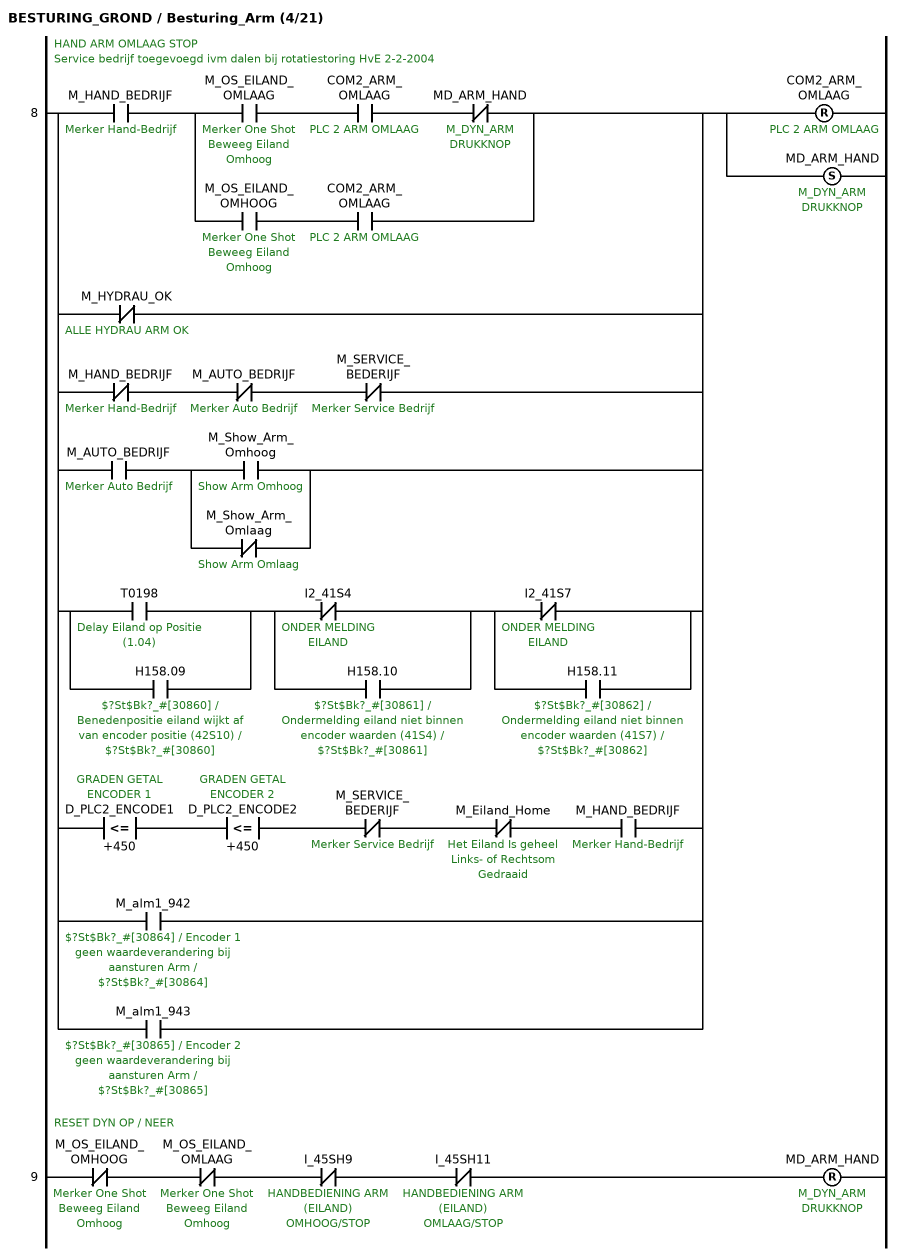
; [picture p373: BESTURING_GROND / Besturing_Arm, rungs 8-9]
; rung 8: HAND ARM OMLAAG STOP / Service bedrijf toegevoegd ivm dalen bij rotatiestoring HvE 2-2-2004
LD M_HAND_BEDRIJF  ; Merker Hand-Bedrijf
LD M_OS_EILAND_OMLAAG  ; Merker One Shot Beweeg Eiland Omhoog
AND COM2_ARM_OMLAAG  ; PLC 2 ARM OMLAAG
ANDNOT MD_ARM_HAND  ; M_DYN_ARM DRUKKNOP
LD M_OS_EILAND_OMHOOG  ; Merker One Shot Beweeg Eiland Omhoog
AND COM2_ARM_OMLAAG  ; PLC 2 ARM OMLAAG
ORLD
ANDLD
ORNOT M_HYDRAU_OK  ; ALLE HYDRAU ARM OK
LDNOT M_HAND_BEDRIJF  ; Merker Hand-Bedrijf
ANDNOT M_AUTO_BEDRIJF  ; Merker Auto Bedrijf
ANDNOT M_SERVICE_BEDERIJF  ; Merker Service Bedrijf
ORLD
LD M_AUTO_BEDRIJF  ; Merker Auto Bedrijf
LD M_Show_Arm_Omhoog  ; Show Arm Omhoog
ORNOT M_Show_Arm_Omlaag  ; Show Arm Omlaag
ANDLD
ORLD
LD T0198  ; Delay Eiland op Positie (1.04)
OR H158.09  ; $?St$Bk?_#[30860] / Benedenpositie eiland wijkt af van encoder positie (42S10) / $?St$Bk?_#[30860]
LDNOT I2_41S4  ; ONDER MELDING EILAND
OR H158.10  ; $?St$Bk?_#[30861] / Ondermelding eiland niet binnen encoder waarden (41S4) / $?St$Bk?_#[30861]
ANDLD
LDNOT I2_41S7  ; ONDER MELDING EILAND
OR H158.11  ; $?St$Bk?_#[30862] / Ondermelding eiland niet binnen encoder waarden (41S7) / $?St$Bk?_#[30862]
ANDLD
ORLD
LD<=S(317) D_PLC2_ENCODE1 +450  ; GRADEN GETAL ENCODER 1
AND<=S(317) D_PLC2_ENCODE2 +450  ; GRADEN GETAL ENCODER 2
ANDNOT M_SERVICE_BEDERIJF  ; Merker Service Bedrijf
ANDNOT M_Eiland_Home  ; Het Eiland Is geheel Links- of Rechtsom Gedraaid
AND M_HAND_BEDRIJF  ; Merker Hand-Bedrijf
ORLD
OR M_alm1_942  ; $?St$Bk?_#[30864] / Encoder 1 geen waardeverandering bij aansturen Arm / $?St$Bk?_#[30864]
OR M_alm1_943  ; $?St$Bk?_#[30865] / Encoder 2 geen waardeverandering bij aansturen Arm / $?St$Bk?_#[30865]
RSET COM2_ARM_OMLAAG  ; PLC 2 ARM OMLAAG
SET MD_ARM_HAND  ; M_DYN_ARM DRUKKNOP
; rung 9: RESET DYN OP / NEER
LDNOT M_OS_EILAND_OMHOOG  ; Merker One Shot Beweeg Eiland Omhoog
ANDNOT M_OS_EILAND_OMLAAG  ; Merker One Shot Beweeg Eiland Omhoog
ANDNOT I_45SH9  ; HANDBEDIENING ARM (EILAND) OMHOOG/STOP
ANDNOT I_45SH11  ; HANDBEDIENING ARM (EILAND) OMLAAG/STOP
RSET MD_ARM_HAND  ; M_DYN_ARM DRUKKNOP

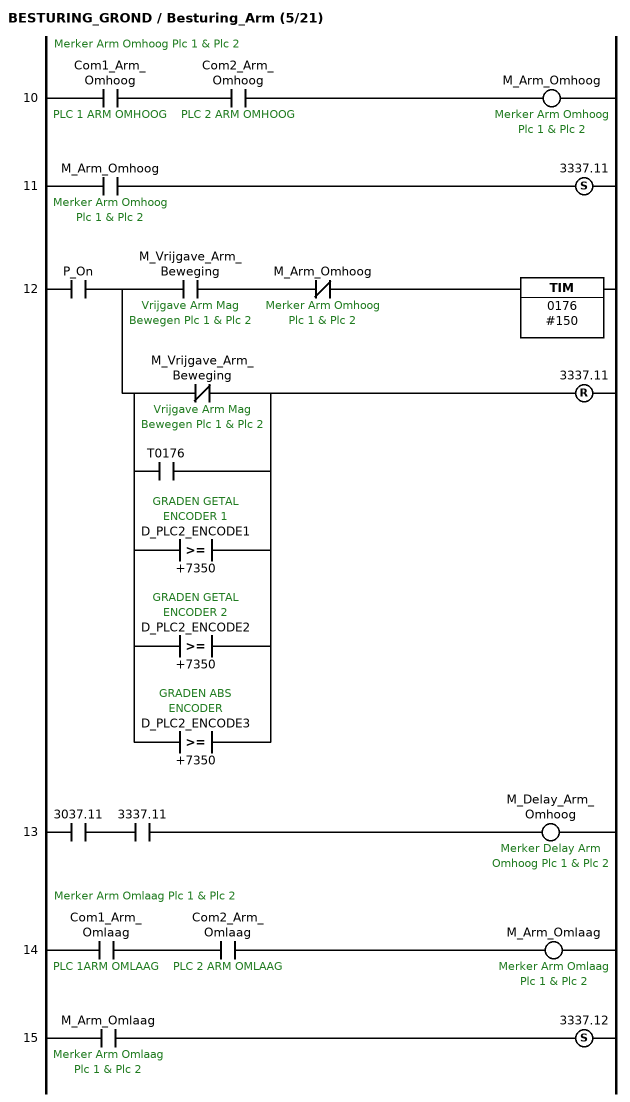
; rung 10: Merker Arm Omhoog Plc 1 & Plc 2
LD Com1_Arm_Omhoog  ; PLC 1 ARM OMHOOG
AND Com2_Arm_Omhoog  ; PLC 2 ARM OMHOOG
OUT M_Arm_Omhoog  ; Merker Arm Omhoog Plc 1 & Plc 2
; rung 11
LD M_Arm_Omhoog  ; Merker Arm Omhoog Plc 1 & Plc 2
SET 3337.11
; rung 12
LD P_On
OUT TR0
AND M_Vrijgave_Arm_Beweging  ; Vrijgave Arm Mag Bewegen Plc 1 & Plc 2
ANDNOT M_Arm_Omhoog  ; Merker Arm Omhoog Plc 1 & Plc 2
TIM 0176 #150
LD TR0
LDNOT M_Vrijgave_Arm_Beweging  ; Vrijgave Arm Mag Bewegen Plc 1 & Plc 2
OR T0176
OR>=S(327) D_PLC2_ENCODE1 +7350  ; GRADEN GETAL ENCODER 1
OR>=S(327) D_PLC2_ENCODE2 +7350  ; GRADEN GETAL ENCODER 2
OR>=S(327) D_PLC2_ENCODE3 +7350  ; GRADEN ABS ENCODER
ANDLD
RSET 3337.11
; rung 13
LD 3037.11
AND 3337.11
OUT M_Delay_Arm_Omhoog  ; Merker Delay Arm Omhoog Plc 1 & Plc 2
; rung 14: Merker Arm Omlaag Plc 1 & Plc 2
LD Com1_Arm_Omlaag  ; PLC 1ARM OMLAAG
AND Com2_Arm_Omlaag  ; PLC 2 ARM OMLAAG
OUT M_Arm_Omlaag  ; Merker Arm Omlaag Plc 1 & Plc 2
; rung 15
LD M_Arm_Omlaag  ; Merker Arm Omlaag Plc 1 & Plc 2
SET 3337.12

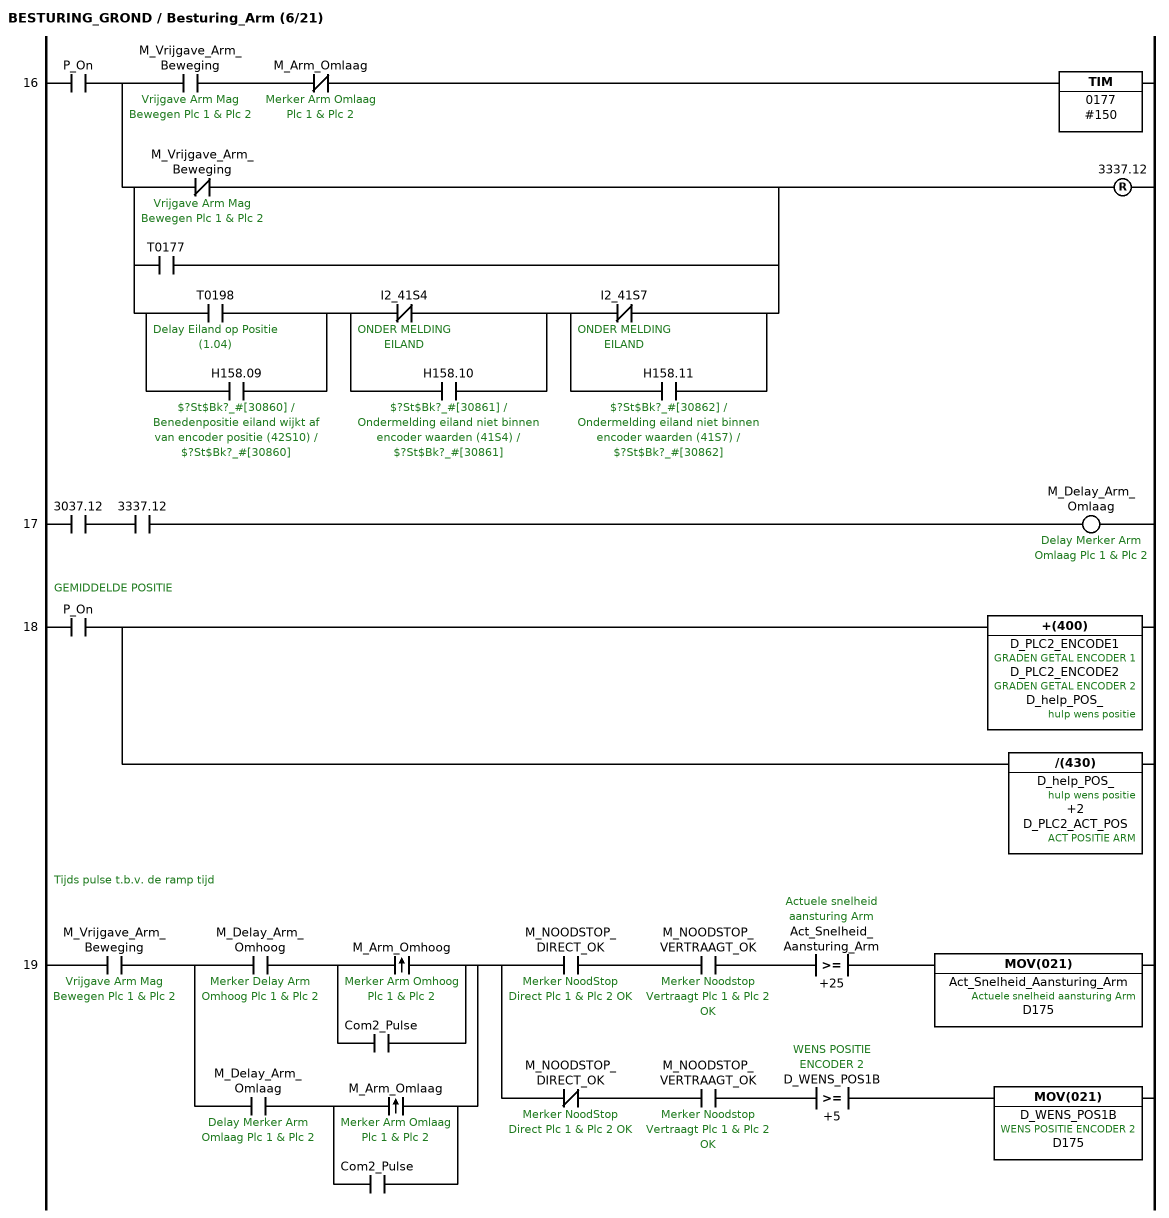
; rung 16
LD P_On
OUT TR0
AND M_Vrijgave_Arm_Beweging  ; Vrijgave Arm Mag Bewegen Plc 1 & Plc 2
ANDNOT M_Arm_Omlaag  ; Merker Arm Omlaag Plc 1 & Plc 2
TIM 0177 #150
LD TR0
LDNOT M_Vrijgave_Arm_Beweging  ; Vrijgave Arm Mag Bewegen Plc 1 & Plc 2
OR T0177
LD T0198  ; Delay Eiland op Positie (1.04)
OR H158.09  ; $?St$Bk?_#[30860] / Benedenpositie eiland wijkt af van encoder positie (42S10) / $?St$Bk?_#[30860]
LDNOT I2_41S4  ; ONDER MELDING EILAND
OR H158.10  ; $?St$Bk?_#[30861] / Ondermelding eiland niet binnen encoder waarden (41S4) / $?St$Bk?_#[30861]
ANDLD
LDNOT I2_41S7  ; ONDER MELDING EILAND
OR H158.11  ; $?St$Bk?_#[30862] / Ondermelding eiland niet binnen encoder waarden (41S7) / $?St$Bk?_#[30862]
ANDLD
ORLD
ANDLD
RSET 3337.12
; rung 17
LD 3037.12
AND 3337.12
OUT M_Delay_Arm_Omlaag  ; Delay Merker Arm Omlaag Plc 1 & Plc 2
; rung 18: GEMIDDELDE POSITIE
LD P_On
+(400) D_PLC2_ENCODE1 D_PLC2_ENCODE2 D_help_POS_  ; GRADEN GETAL ENCODER 1, GRADEN GETAL ENCODER 2, hulp wens positie
/(430) D_help_POS_ +2 D_PLC2_ACT_POS  ; hulp wens positie, ACT POSITIE ARM
; rung 19: Tijds pulse t.b.v. de ramp tijd
LD M_Vrijgave_Arm_Beweging  ; Vrijgave Arm Mag Bewegen Plc 1 & Plc 2
LD M_Delay_Arm_Omhoog  ; Merker Delay Arm Omhoog Plc 1 & Plc 2
@LD M_Arm_Omhoog  ; Merker Arm Omhoog Plc 1 & Plc 2
OR Com2_Pulse
ANDLD
LD M_Delay_Arm_Omlaag  ; Delay Merker Arm Omlaag Plc 1 & Plc 2
@LD M_Arm_Omlaag  ; Merker Arm Omlaag Plc 1 & Plc 2
OR Com2_Pulse
ANDLD
ORLD
ANDLD
OUT TR0
AND M_NOODSTOP_DIRECT_OK  ; Merker NoodStop Direct Plc 1 & Plc 2 OK
AND M_NOODSTOP_VERTRAAGT_OK  ; Merker Noodstop Vertraagt Plc 1 & Plc 2 OK
AND>=S(327) Act_Snelheid_Aansturing_Arm +25  ; Actuele snelheid aansturing Arm
MOV(021) Act_Snelheid_Aansturing_Arm D175  ; Actuele snelheid aansturing Arm
LD TR0
ANDNOT M_NOODSTOP_DIRECT_OK  ; Merker NoodStop Direct Plc 1 & Plc 2 OK
AND M_NOODSTOP_VERTRAAGT_OK  ; Merker Noodstop Vertraagt Plc 1 & Plc 2 OK
AND>=S(327) D_WENS_POS1B +5  ; WENS POSITIE ENCODER 2
MOV(021) D_WENS_POS1B D175  ; WENS POSITIE ENCODER 2

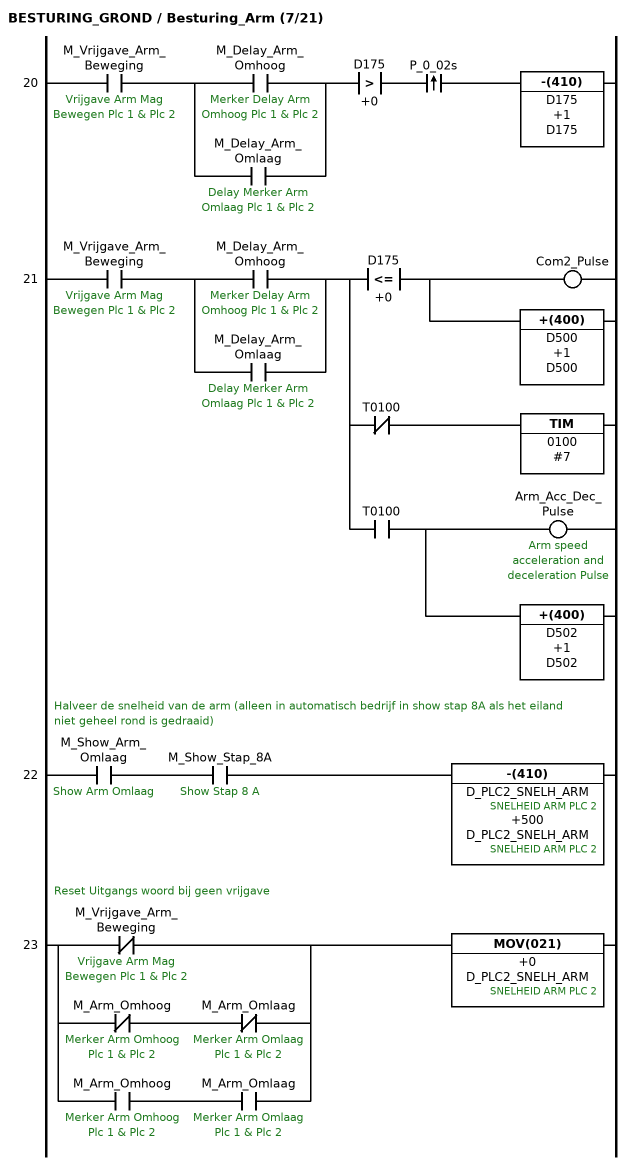
; rung 20
LD M_Vrijgave_Arm_Beweging  ; Vrijgave Arm Mag Bewegen Plc 1 & Plc 2
LD M_Delay_Arm_Omhoog  ; Merker Delay Arm Omhoog Plc 1 & Plc 2
OR M_Delay_Arm_Omlaag  ; Delay Merker Arm Omlaag Plc 1 & Plc 2
ANDLD
AND>S(322) D175 +0
@AND P_0_02s
-(410) D175 +1 D175
; rung 21
LD M_Vrijgave_Arm_Beweging  ; Vrijgave Arm Mag Bewegen Plc 1 & Plc 2
LD M_Delay_Arm_Omhoog  ; Merker Delay Arm Omhoog Plc 1 & Plc 2
OR M_Delay_Arm_Omlaag  ; Delay Merker Arm Omlaag Plc 1 & Plc 2
ANDLD
OUT TR0
AND<=S(317) D175 +0
OUT Com2_Pulse
+(400) D500 +1 D500
LD TR0
ANDNOT T0100
TIM 0100 #7
LD TR0
AND T0100
OUT Arm_Acc_Dec_Pulse  ; Arm speed acceleration and deceleration Pulse
+(400) D502 +1 D502
; rung 22: Halveer de snelheid van de arm (alleen in automatisch bedrijf in show stap 8A als het eiland niet geheel rond is gedraaid)
LD M_Show_Arm_Omlaag  ; Show Arm Omlaag
AND M_Show_Stap_8A  ; Show Stap 8 A
-(410) D_PLC2_SNELH_ARM +500 D_PLC2_SNELH_ARM  ; SNELHEID ARM PLC 2
; rung 23: Reset Uitgangs woord bij geen vrijgave
LDNOT M_Vrijgave_Arm_Beweging  ; Vrijgave Arm Mag Bewegen Plc 1 & Plc 2
LDNOT M_Arm_Omhoog  ; Merker Arm Omhoog Plc 1 & Plc 2
ANDNOT M_Arm_Omlaag  ; Merker Arm Omlaag Plc 1 & Plc 2
ORLD
LD M_Arm_Omhoog  ; Merker Arm Omhoog Plc 1 & Plc 2
AND M_Arm_Omlaag  ; Merker Arm Omlaag Plc 1 & Plc 2
ORLD
MOV(021) +0 D_PLC2_SNELH_ARM  ; SNELHEID ARM PLC 2

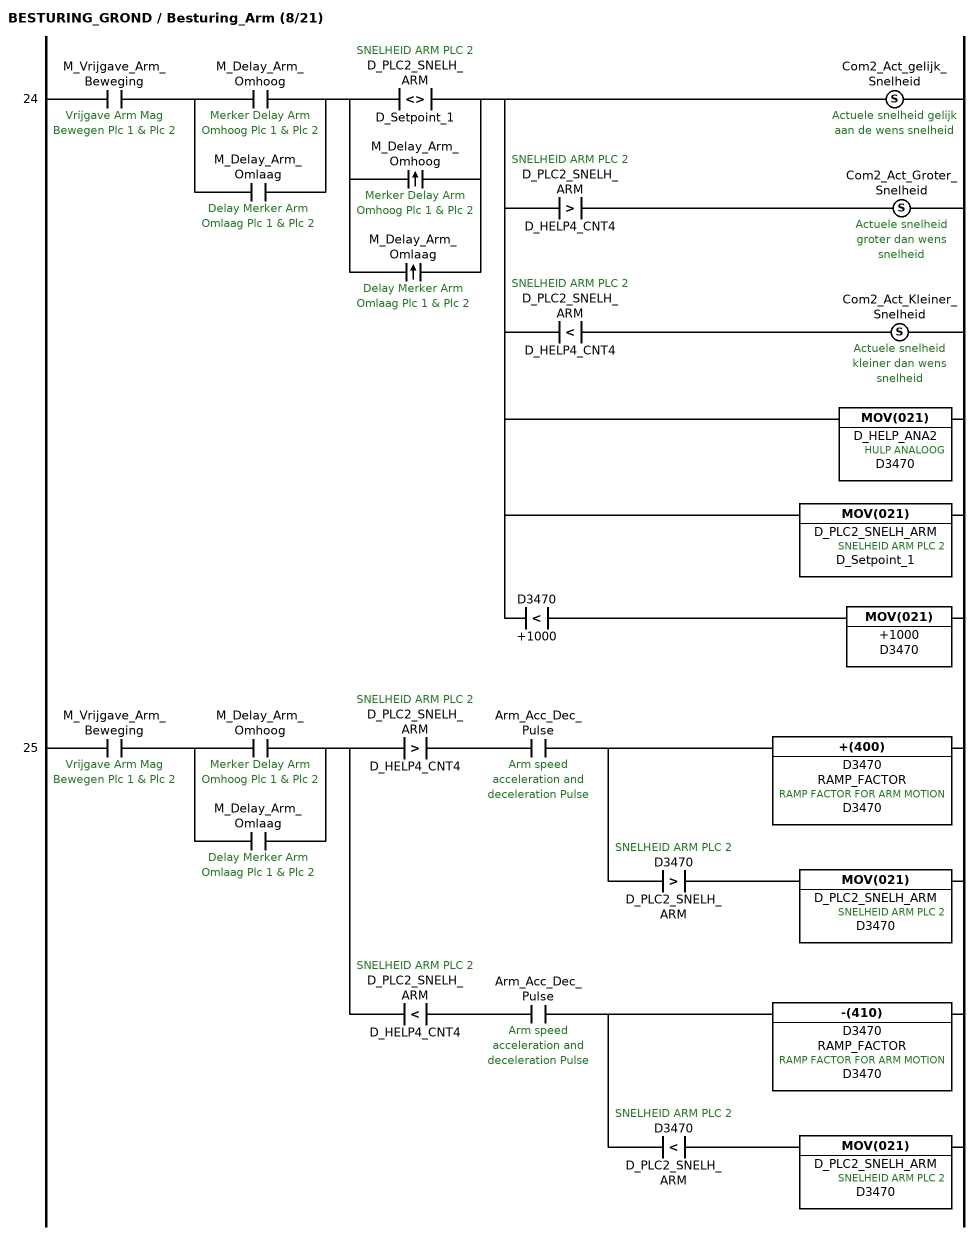
; rung 24
LD M_Vrijgave_Arm_Beweging  ; Vrijgave Arm Mag Bewegen Plc 1 & Plc 2
LD M_Delay_Arm_Omhoog  ; Merker Delay Arm Omhoog Plc 1 & Plc 2
OR M_Delay_Arm_Omlaag  ; Delay Merker Arm Omlaag Plc 1 & Plc 2
ANDLD
LD<>(305) D_PLC2_SNELH_ARM D_Setpoint_1  ; SNELHEID ARM PLC 2
@OR M_Delay_Arm_Omhoog  ; Merker Delay Arm Omhoog Plc 1 & Plc 2
@OR M_Delay_Arm_Omlaag  ; Delay Merker Arm Omlaag Plc 1 & Plc 2
ANDLD
OUT TR0
SET Com2_Act_gelijk_Snelheid  ; Actuele snelheid gelijk aan de wens snelheid
AND>(320) D_PLC2_SNELH_ARM D_HELP4_CNT4  ; SNELHEID ARM PLC 2
SET Com2_Act_Groter_Snelheid  ; Actuele snelheid groter dan wens snelheid
LD TR0
AND<(310) D_PLC2_SNELH_ARM D_HELP4_CNT4  ; SNELHEID ARM PLC 2
SET Com2_Act_Kleiner_Snelheid  ; Actuele snelheid kleiner dan wens snelheid
LD TR0
MOV(021) D_HELP_ANA2 D3470  ; HULP ANALOOG
MOV(021) D_PLC2_SNELH_ARM D_Setpoint_1  ; SNELHEID ARM PLC 2
AND<S(312) D3470 +1000
MOV(021) +1000 D3470
; rung 25
LD M_Vrijgave_Arm_Beweging  ; Vrijgave Arm Mag Bewegen Plc 1 & Plc 2
LD M_Delay_Arm_Omhoog  ; Merker Delay Arm Omhoog Plc 1 & Plc 2
OR M_Delay_Arm_Omlaag  ; Delay Merker Arm Omlaag Plc 1 & Plc 2
ANDLD
OUT TR0
AND>(320) D_PLC2_SNELH_ARM D_HELP4_CNT4  ; SNELHEID ARM PLC 2
AND Arm_Acc_Dec_Pulse  ; Arm speed acceleration and deceleration Pulse
+(400) D3470 RAMP_FACTOR D3470  ; RAMP FACTOR FOR ARM MOTION
AND>(320) D3470 D_PLC2_SNELH_ARM  ; SNELHEID ARM PLC 2
MOV(021) D_PLC2_SNELH_ARM D3470  ; SNELHEID ARM PLC 2
LD TR0
AND<(310) D_PLC2_SNELH_ARM D_HELP4_CNT4  ; SNELHEID ARM PLC 2
AND Arm_Acc_Dec_Pulse  ; Arm speed acceleration and deceleration Pulse
-(410) D3470 RAMP_FACTOR D3470  ; RAMP FACTOR FOR ARM MOTION
AND<(310) D3470 D_PLC2_SNELH_ARM  ; SNELHEID ARM PLC 2
MOV(021) D_PLC2_SNELH_ARM D3470  ; SNELHEID ARM PLC 2

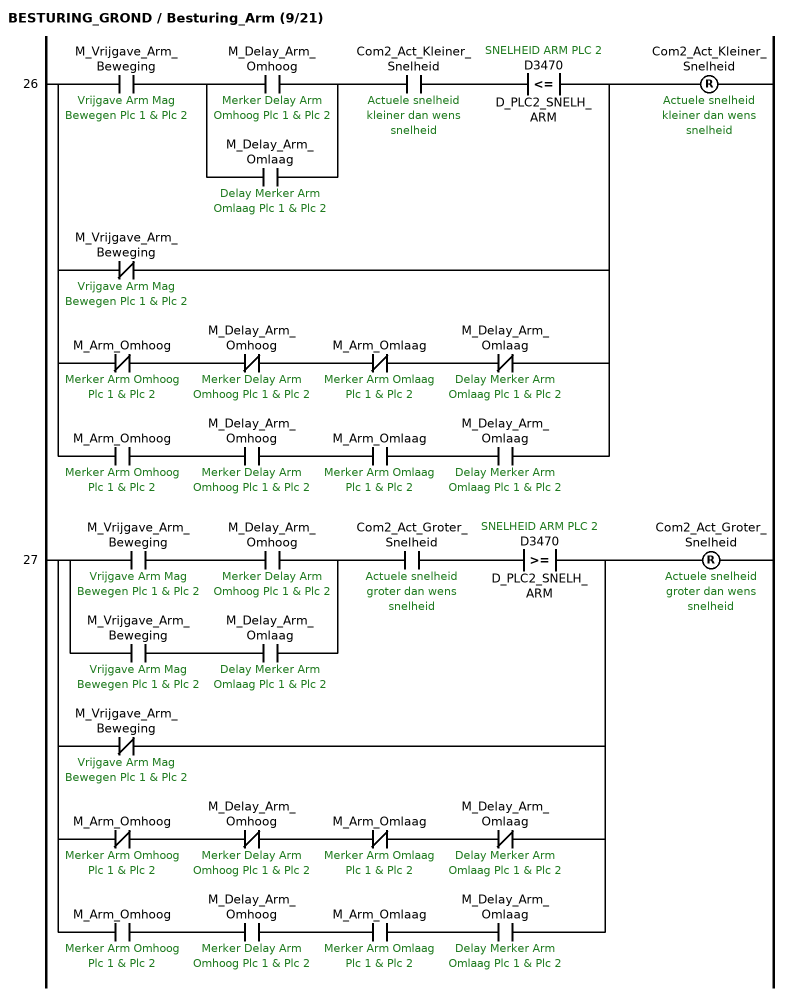
; rung 26
LD M_Vrijgave_Arm_Beweging  ; Vrijgave Arm Mag Bewegen Plc 1 & Plc 2
LD M_Delay_Arm_Omhoog  ; Merker Delay Arm Omhoog Plc 1 & Plc 2
OR M_Delay_Arm_Omlaag  ; Delay Merker Arm Omlaag Plc 1 & Plc 2
ANDLD
AND Com2_Act_Kleiner_Snelheid  ; Actuele snelheid kleiner dan wens snelheid
AND<=(315) D3470 D_PLC2_SNELH_ARM  ; SNELHEID ARM PLC 2
ORNOT M_Vrijgave_Arm_Beweging  ; Vrijgave Arm Mag Bewegen Plc 1 & Plc 2
LDNOT M_Arm_Omhoog  ; Merker Arm Omhoog Plc 1 & Plc 2
ANDNOT M_Delay_Arm_Omhoog  ; Merker Delay Arm Omhoog Plc 1 & Plc 2
ANDNOT M_Arm_Omlaag  ; Merker Arm Omlaag Plc 1 & Plc 2
ANDNOT M_Delay_Arm_Omlaag  ; Delay Merker Arm Omlaag Plc 1 & Plc 2
ORLD
LD M_Arm_Omhoog  ; Merker Arm Omhoog Plc 1 & Plc 2
AND M_Delay_Arm_Omhoog  ; Merker Delay Arm Omhoog Plc 1 & Plc 2
AND M_Arm_Omlaag  ; Merker Arm Omlaag Plc 1 & Plc 2
AND M_Delay_Arm_Omlaag  ; Delay Merker Arm Omlaag Plc 1 & Plc 2
ORLD
RSET Com2_Act_Kleiner_Snelheid  ; Actuele snelheid kleiner dan wens snelheid
; rung 27
LD M_Vrijgave_Arm_Beweging  ; Vrijgave Arm Mag Bewegen Plc 1 & Plc 2
AND M_Delay_Arm_Omhoog  ; Merker Delay Arm Omhoog Plc 1 & Plc 2
LD M_Vrijgave_Arm_Beweging  ; Vrijgave Arm Mag Bewegen Plc 1 & Plc 2
AND M_Delay_Arm_Omlaag  ; Delay Merker Arm Omlaag Plc 1 & Plc 2
ORLD
AND Com2_Act_Groter_Snelheid  ; Actuele snelheid groter dan wens snelheid
AND>=(325) D3470 D_PLC2_SNELH_ARM  ; SNELHEID ARM PLC 2
ORNOT M_Vrijgave_Arm_Beweging  ; Vrijgave Arm Mag Bewegen Plc 1 & Plc 2
LDNOT M_Arm_Omhoog  ; Merker Arm Omhoog Plc 1 & Plc 2
ANDNOT M_Delay_Arm_Omhoog  ; Merker Delay Arm Omhoog Plc 1 & Plc 2
ANDNOT M_Arm_Omlaag  ; Merker Arm Omlaag Plc 1 & Plc 2
ANDNOT M_Delay_Arm_Omlaag  ; Delay Merker Arm Omlaag Plc 1 & Plc 2
ORLD
LD M_Arm_Omhoog  ; Merker Arm Omhoog Plc 1 & Plc 2
AND M_Delay_Arm_Omhoog  ; Merker Delay Arm Omhoog Plc 1 & Plc 2
AND M_Arm_Omlaag  ; Merker Arm Omlaag Plc 1 & Plc 2
AND M_Delay_Arm_Omlaag  ; Delay Merker Arm Omlaag Plc 1 & Plc 2
ORLD
RSET Com2_Act_Groter_Snelheid  ; Actuele snelheid groter dan wens snelheid

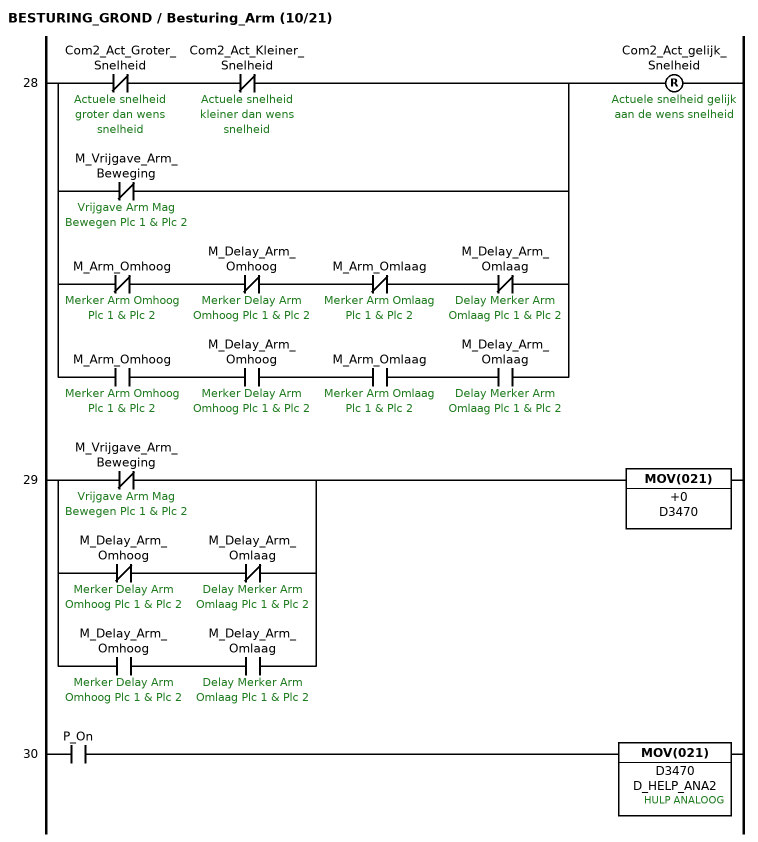
; rung 28
LDNOT Com2_Act_Groter_Snelheid  ; Actuele snelheid groter dan wens snelheid
ANDNOT Com2_Act_Kleiner_Snelheid  ; Actuele snelheid kleiner dan wens snelheid
ORNOT M_Vrijgave_Arm_Beweging  ; Vrijgave Arm Mag Bewegen Plc 1 & Plc 2
LDNOT M_Arm_Omhoog  ; Merker Arm Omhoog Plc 1 & Plc 2
ANDNOT M_Delay_Arm_Omhoog  ; Merker Delay Arm Omhoog Plc 1 & Plc 2
ANDNOT M_Arm_Omlaag  ; Merker Arm Omlaag Plc 1 & Plc 2
ANDNOT M_Delay_Arm_Omlaag  ; Delay Merker Arm Omlaag Plc 1 & Plc 2
ORLD
LD M_Arm_Omhoog  ; Merker Arm Omhoog Plc 1 & Plc 2
AND M_Delay_Arm_Omhoog  ; Merker Delay Arm Omhoog Plc 1 & Plc 2
AND M_Arm_Omlaag  ; Merker Arm Omlaag Plc 1 & Plc 2
AND M_Delay_Arm_Omlaag  ; Delay Merker Arm Omlaag Plc 1 & Plc 2
ORLD
RSET Com2_Act_gelijk_Snelheid  ; Actuele snelheid gelijk aan de wens snelheid
; rung 29
LDNOT M_Vrijgave_Arm_Beweging  ; Vrijgave Arm Mag Bewegen Plc 1 & Plc 2
LDNOT M_Delay_Arm_Omhoog  ; Merker Delay Arm Omhoog Plc 1 & Plc 2
ANDNOT M_Delay_Arm_Omlaag  ; Delay Merker Arm Omlaag Plc 1 & Plc 2
ORLD
LD M_Delay_Arm_Omhoog  ; Merker Delay Arm Omhoog Plc 1 & Plc 2
AND M_Delay_Arm_Omlaag  ; Delay Merker Arm Omlaag Plc 1 & Plc 2
ORLD
MOV(021) +0 D3470
; rung 30
LD P_On
MOV(021) D3470 D_HELP_ANA2  ; HULP ANALOOG

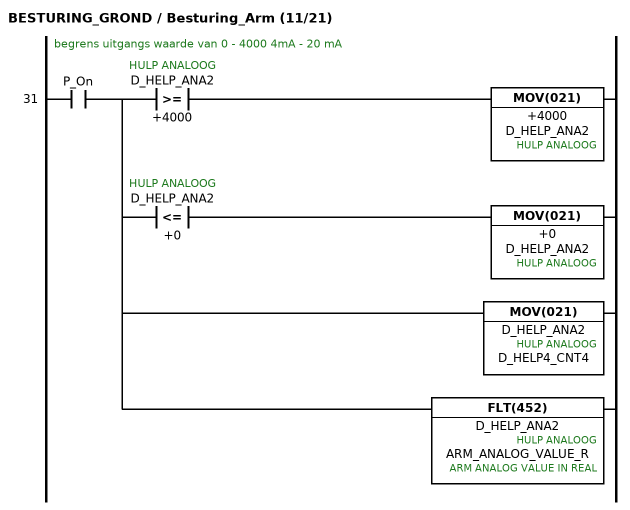
; rung 31: begrens uitgangs waarde van 0 - 4000 4mA - 20 mA
LD P_On
OUT TR0
AND>=S(327) D_HELP_ANA2 +4000  ; HULP ANALOOG
MOV(021) +4000 D_HELP_ANA2  ; HULP ANALOOG
LD TR0
AND<=S(317) D_HELP_ANA2 +0  ; HULP ANALOOG
MOV(021) +0 D_HELP_ANA2  ; HULP ANALOOG
LD TR0
MOV(021) D_HELP_ANA2 D_HELP4_CNT4  ; HULP ANALOOG
FLT(452) D_HELP_ANA2 ARM_ANALOG_VALUE_R  ; HULP ANALOOG, ARM ANALOG VALUE IN REAL

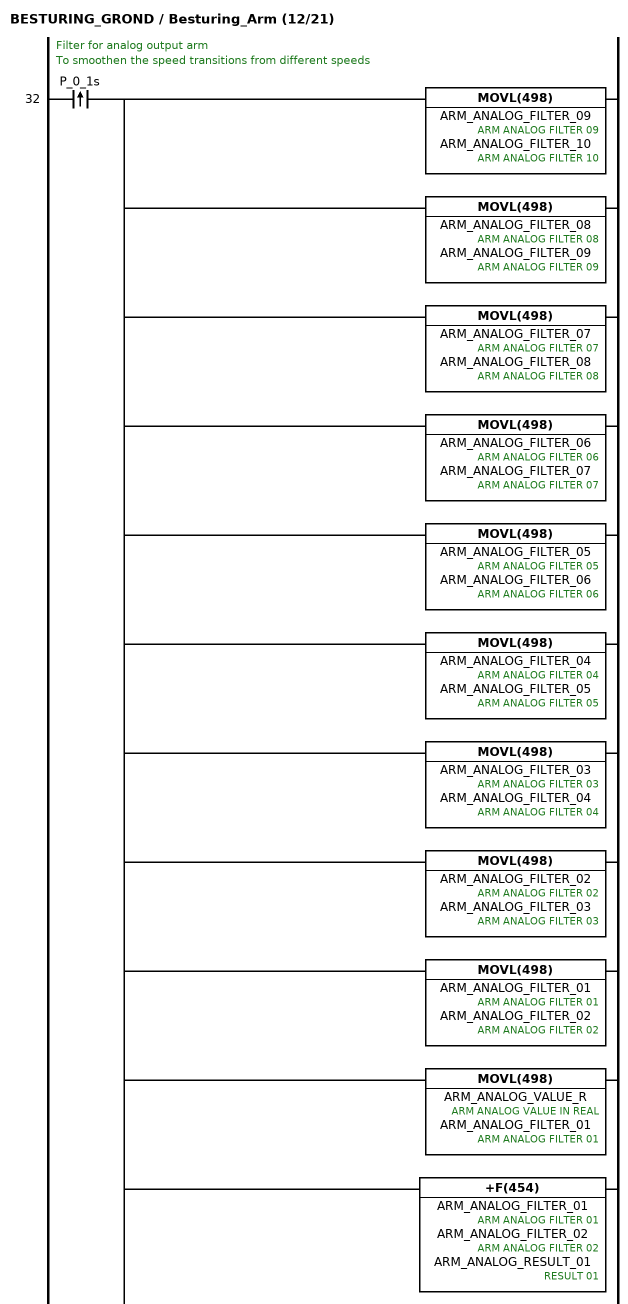

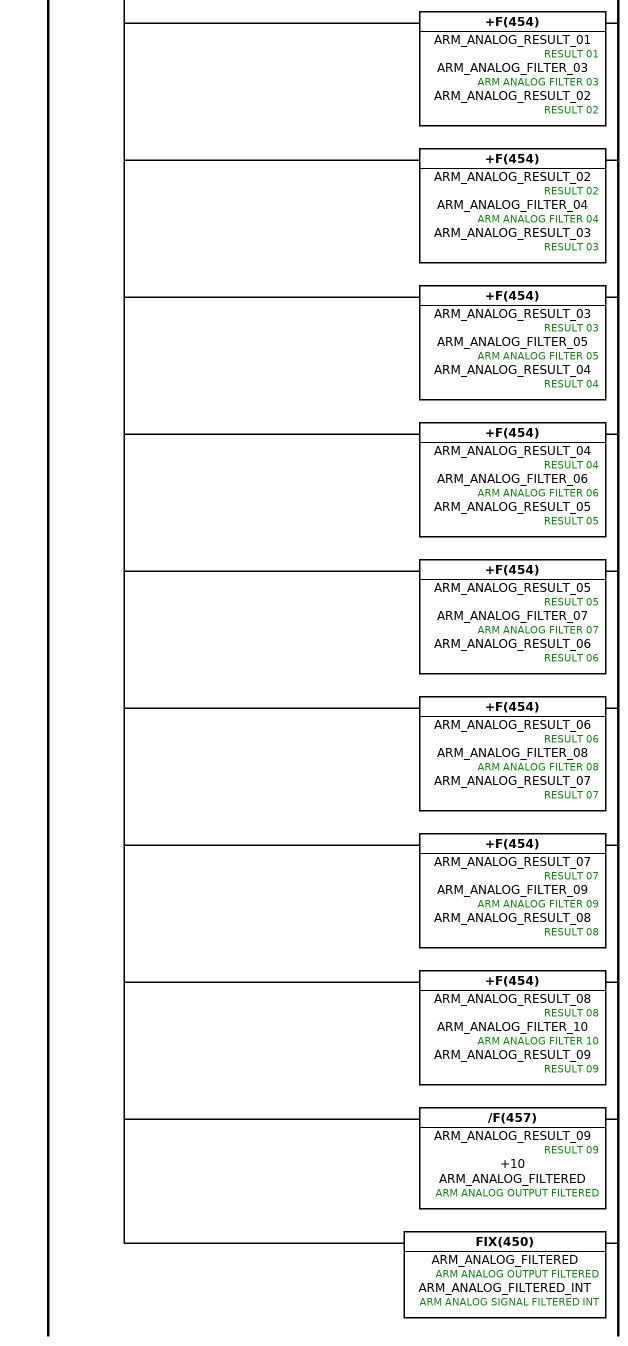
; rung 32: Filter for analog output arm / To smoothen the speed transitions from different speeds
@LD P_0_1s
MOVL(498) ARM_ANALOG_FILTER_09 ARM_ANALOG_FILTER_10  ; ARM ANALOG FILTER 09, ARM ANALOG FILTER 10
MOVL(498) ARM_ANALOG_FILTER_08 ARM_ANALOG_FILTER_09  ; ARM ANALOG FILTER 08, ARM ANALOG FILTER 09
MOVL(498) ARM_ANALOG_FILTER_07 ARM_ANALOG_FILTER_08  ; ARM ANALOG FILTER 07, ARM ANALOG FILTER 08
MOVL(498) ARM_ANALOG_FILTER_06 ARM_ANALOG_FILTER_07  ; ARM ANALOG FILTER 06, ARM ANALOG FILTER 07
MOVL(498) ARM_ANALOG_FILTER_05 ARM_ANALOG_FILTER_06  ; ARM ANALOG FILTER 05, ARM ANALOG FILTER 06
MOVL(498) ARM_ANALOG_FILTER_04 ARM_ANALOG_FILTER_05  ; ARM ANALOG FILTER 04, ARM ANALOG FILTER 05
MOVL(498) ARM_ANALOG_FILTER_03 ARM_ANALOG_FILTER_04  ; ARM ANALOG FILTER 03, ARM ANALOG FILTER 04
MOVL(498) ARM_ANALOG_FILTER_02 ARM_ANALOG_FILTER_03  ; ARM ANALOG FILTER 02, ARM ANALOG FILTER 03
MOVL(498) ARM_ANALOG_FILTER_01 ARM_ANALOG_FILTER_02  ; ARM ANALOG FILTER 01, ARM ANALOG FILTER 02
MOVL(498) ARM_ANALOG_VALUE_R ARM_ANALOG_FILTER_01  ; ARM ANALOG VALUE IN REAL, ARM ANALOG FILTER 01
+F(454) ARM_ANALOG_FILTER_01 ARM_ANALOG_FILTER_02 ARM_ANALOG_RESULT_01  ; ARM ANALOG FILTER 01, ARM ANALOG FILTER 02, RESULT 01
+F(454) ARM_ANALOG_RESULT_01 ARM_ANALOG_FILTER_03 ARM_ANALOG_RESULT_02  ; RESULT 01, ARM ANALOG FILTER 03, RESULT 02
+F(454) ARM_ANALOG_RESULT_02 ARM_ANALOG_FILTER_04 ARM_ANALOG_RESULT_03  ; RESULT 02, ARM ANALOG FILTER 04, RESULT 03
+F(454) ARM_ANALOG_RESULT_03 ARM_ANALOG_FILTER_05 ARM_ANALOG_RESULT_04  ; RESULT 03, ARM ANALOG FILTER 05, RESULT 04
+F(454) ARM_ANALOG_RESULT_04 ARM_ANALOG_FILTER_06 ARM_ANALOG_RESULT_05  ; RESULT 04, ARM ANALOG FILTER 06, RESULT 05
+F(454) ARM_ANALOG_RESULT_05 ARM_ANALOG_FILTER_07 ARM_ANALOG_RESULT_06  ; RESULT 05, ARM ANALOG FILTER 07, RESULT 06
+F(454) ARM_ANALOG_RESULT_06 ARM_ANALOG_FILTER_08 ARM_ANALOG_RESULT_07  ; RESULT 06, ARM ANALOG FILTER 08, RESULT 07
+F(454) ARM_ANALOG_RESULT_07 ARM_ANALOG_FILTER_09 ARM_ANALOG_RESULT_08  ; RESULT 07, ARM ANALOG FILTER 09, RESULT 08
+F(454) ARM_ANALOG_RESULT_08 ARM_ANALOG_FILTER_10 ARM_ANALOG_RESULT_09  ; RESULT 08, ARM ANALOG FILTER 10, RESULT 09
/F(457) ARM_ANALOG_RESULT_09 +10 ARM_ANALOG_FILTERED  ; RESULT 09, ARM ANALOG OUTPUT FILTERED
FIX(450) ARM_ANALOG_FILTERED ARM_ANALOG_FILTERED_INT  ; ARM ANALOG OUTPUT FILTERED, ARM ANALOG SIGNAL FILTERED INT

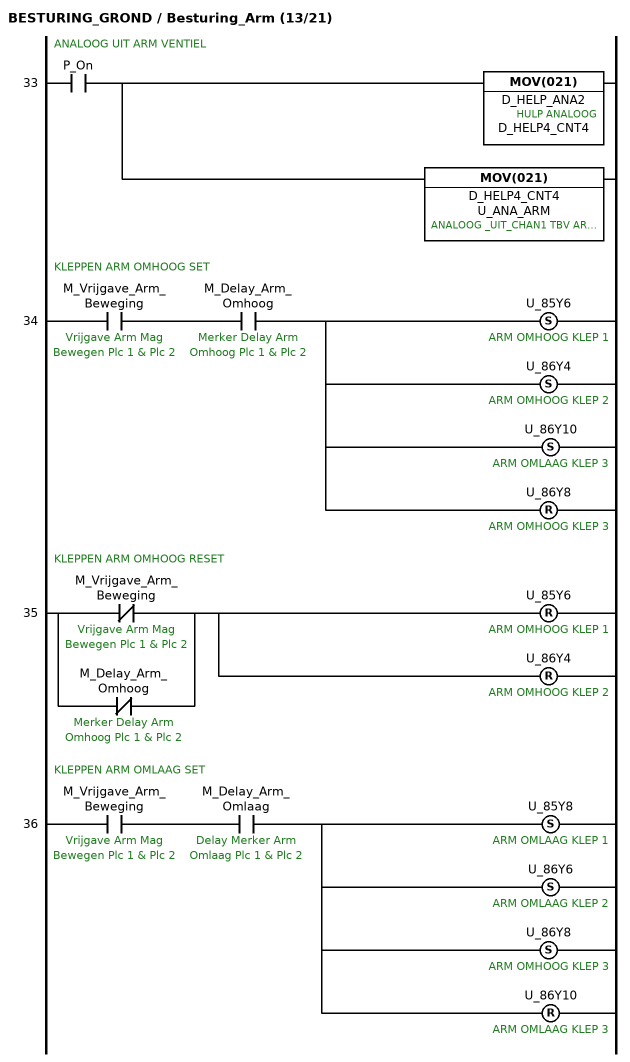
; rung 33: ANALOOG UIT ARM VENTIEL
LD P_On
MOV(021) D_HELP_ANA2 D_HELP4_CNT4  ; HULP ANALOOG
MOV(021) D_HELP4_CNT4 U_ANA_ARM  ; ANALOOG _UIT_CHAN1 TBV ARM BESTURING
; rung 34: KLEPPEN ARM OMHOOG SET
LD M_Vrijgave_Arm_Beweging  ; Vrijgave Arm Mag Bewegen Plc 1 & Plc 2
AND M_Delay_Arm_Omhoog  ; Merker Delay Arm Omhoog Plc 1 & Plc 2
SET U_85Y6  ; ARM OMHOOG KLEP 1
SET U_86Y4  ; ARM OMHOOG KLEP 2
SET U_86Y10  ; ARM OMLAAG KLEP 3
RSET U_86Y8  ; ARM OMHOOG KLEP 3
; rung 35: KLEPPEN ARM OMHOOG RESET
LDNOT M_Vrijgave_Arm_Beweging  ; Vrijgave Arm Mag Bewegen Plc 1 & Plc 2
ORNOT M_Delay_Arm_Omhoog  ; Merker Delay Arm Omhoog Plc 1 & Plc 2
RSET U_85Y6  ; ARM OMHOOG KLEP 1
RSET U_86Y4  ; ARM OMHOOG KLEP 2
; rung 36: KLEPPEN ARM OMLAAG SET
LD M_Vrijgave_Arm_Beweging  ; Vrijgave Arm Mag Bewegen Plc 1 & Plc 2
AND M_Delay_Arm_Omlaag  ; Delay Merker Arm Omlaag Plc 1 & Plc 2
SET U_85Y8  ; ARM OMLAAG KLEP 1
SET U_86Y6  ; ARM OMLAAG KLEP 2
SET U_86Y8  ; ARM OMHOOG KLEP 3
RSET U_86Y10  ; ARM OMLAAG KLEP 3

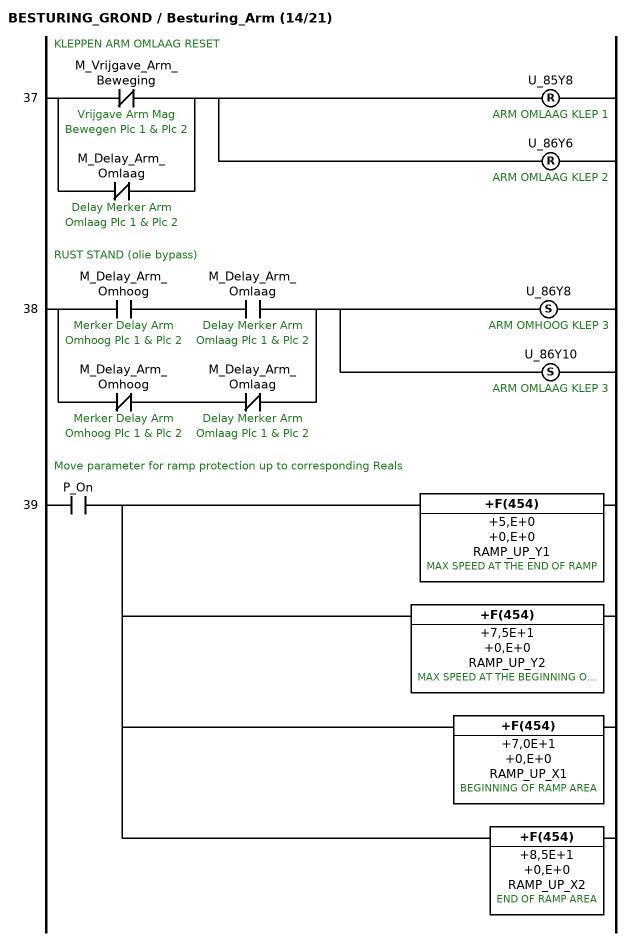
; rung 37: KLEPPEN ARM OMLAAG RESET
LDNOT M_Vrijgave_Arm_Beweging  ; Vrijgave Arm Mag Bewegen Plc 1 & Plc 2
ORNOT M_Delay_Arm_Omlaag  ; Delay Merker Arm Omlaag Plc 1 & Plc 2
RSET U_85Y8  ; ARM OMLAAG KLEP 1
RSET U_86Y6  ; ARM OMLAAG KLEP 2
; rung 38: RUST STAND (olie bypass)
LD M_Delay_Arm_Omhoog  ; Merker Delay Arm Omhoog Plc 1 & Plc 2
AND M_Delay_Arm_Omlaag  ; Delay Merker Arm Omlaag Plc 1 & Plc 2
LDNOT M_Delay_Arm_Omhoog  ; Merker Delay Arm Omhoog Plc 1 & Plc 2
ANDNOT M_Delay_Arm_Omlaag  ; Delay Merker Arm Omlaag Plc 1 & Plc 2
ORLD
SET U_86Y8  ; ARM OMHOOG KLEP 3
SET U_86Y10  ; ARM OMLAAG KLEP 3
; rung 39: Move parameter for ramp protection up to corresponding Reals
LD P_On
+F(454) +5,E+0 +0,E+0 RAMP_UP_Y1  ; MAX SPEED AT THE END OF RAMP
+F(454) +7,5E+1 +0,E+0 RAMP_UP_Y2  ; MAX SPEED AT THE BEGINNING OF RAMP
+F(454) +7,0E+1 +0,E+0 RAMP_UP_X1  ; BEGINNING OF RAMP AREA
+F(454) +8,5E+1 +0,E+0 RAMP_UP_X2  ; END OF RAMP AREA

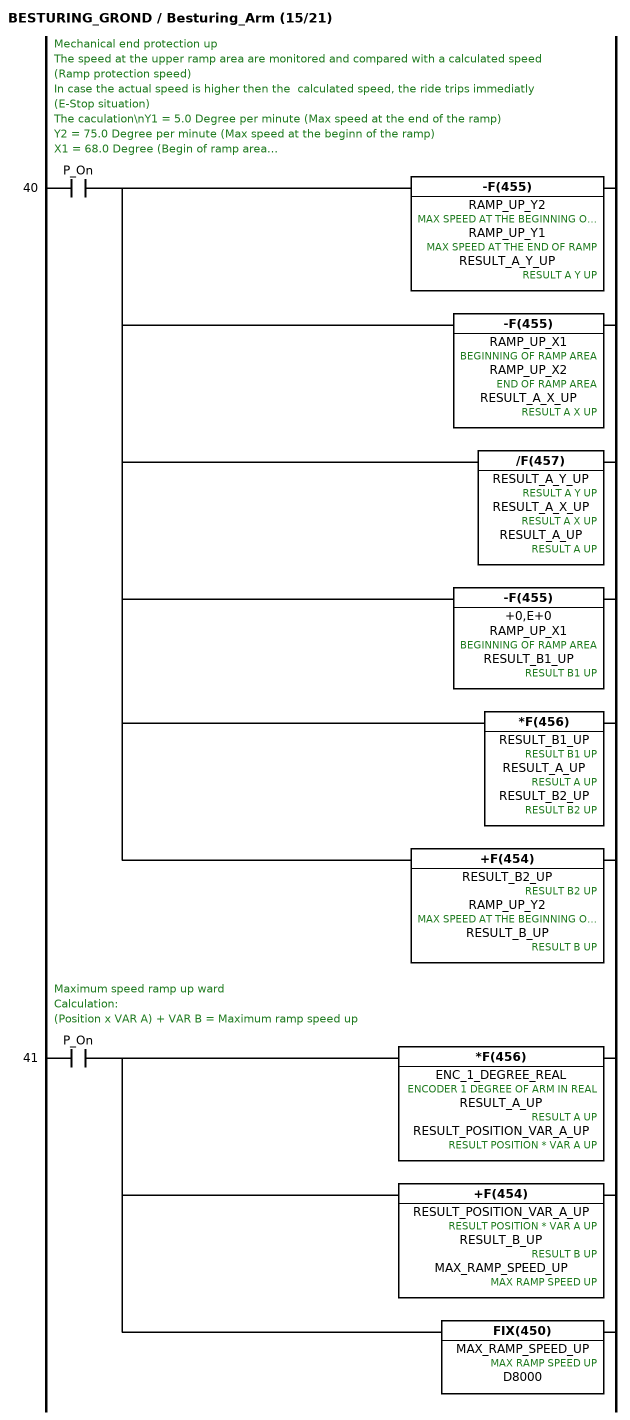
; rung 40: Mechanical end protection up / The speed at the upper ramp area are monitored and compared with a calculated speed (Ramp protection speed) / In case the actual speed is higher then the  calculated speed, the ride trips immediatly (E-Stop situation) / The caculation\nY1 = 5.0 Degree per minute (Max speed at the end of the ramp) / Y2 = 75.0 Degree per minute (Max speed at the beginn of the ramp) / X1 = 68.0 Degree (Begin of ramp area) / X2 = 85.0 Degree (End of ramp area) / The formula for A: / Y2 - Y1 / A =    ------- / X1 - X2 / The formula for B: / B =    (A * (0 - X1) + Y2
LD P_On
-F(455) RAMP_UP_Y2 RAMP_UP_Y1 RESULT_A_Y_UP  ; MAX SPEED AT THE BEGINNING OF RAMP, MAX SPEED AT THE END OF RAMP, RESULT A Y UP
-F(455) RAMP_UP_X1 RAMP_UP_X2 RESULT_A_X_UP  ; BEGINNING OF RAMP AREA, END OF RAMP AREA, RESULT A X UP
/F(457) RESULT_A_Y_UP RESULT_A_X_UP RESULT_A_UP  ; RESULT A Y UP, RESULT A X UP, RESULT A UP
-F(455) +0,E+0 RAMP_UP_X1 RESULT_B1_UP  ; BEGINNING OF RAMP AREA, RESULT B1 UP
*F(456) RESULT_B1_UP RESULT_A_UP RESULT_B2_UP  ; RESULT B1 UP, RESULT A UP, RESULT B2 UP
+F(454) RESULT_B2_UP RAMP_UP_Y2 RESULT_B_UP  ; RESULT B2 UP, MAX SPEED AT THE BEGINNING OF RAMP, RESULT B UP
; rung 41: Maximum speed ramp up ward / Calculation: / (Position x VAR A) + VAR B = Maximum ramp speed up
LD P_On
*F(456) ENC_1_DEGREE_REAL RESULT_A_UP RESULT_POSITION_VAR_A_UP  ; ENCODER 1 DEGREE OF ARM IN REAL, RESULT A UP, RESULT POSITION * VAR A UP
+F(454) RESULT_POSITION_VAR_A_UP RESULT_B_UP MAX_RAMP_SPEED_UP  ; RESULT POSITION * VAR A UP, RESULT B UP, MAX RAMP SPEED UP
FIX(450) MAX_RAMP_SPEED_UP D8000  ; MAX RAMP SPEED UP

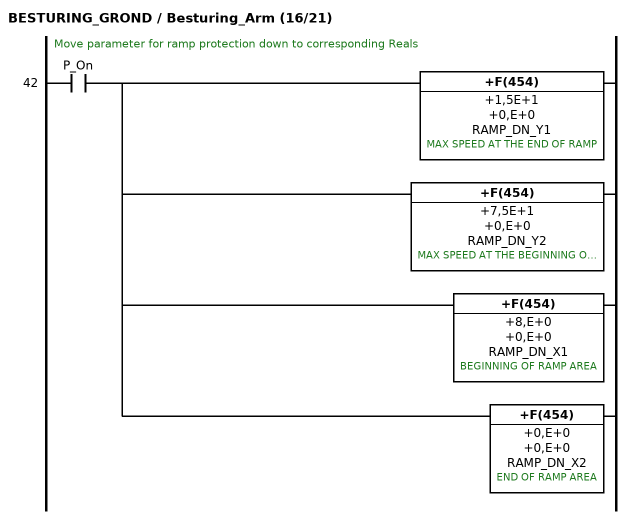
; rung 42: Move parameter for ramp protection down to corresponding Reals
LD P_On
+F(454) +1,5E+1 +0,E+0 RAMP_DN_Y1  ; MAX SPEED AT THE END OF RAMP
+F(454) +7,5E+1 +0,E+0 RAMP_DN_Y2  ; MAX SPEED AT THE BEGINNING OF RAMP
+F(454) +8,E+0 +0,E+0 RAMP_DN_X1  ; BEGINNING OF RAMP AREA
+F(454) +0,E+0 +0,E+0 RAMP_DN_X2  ; END OF RAMP AREA

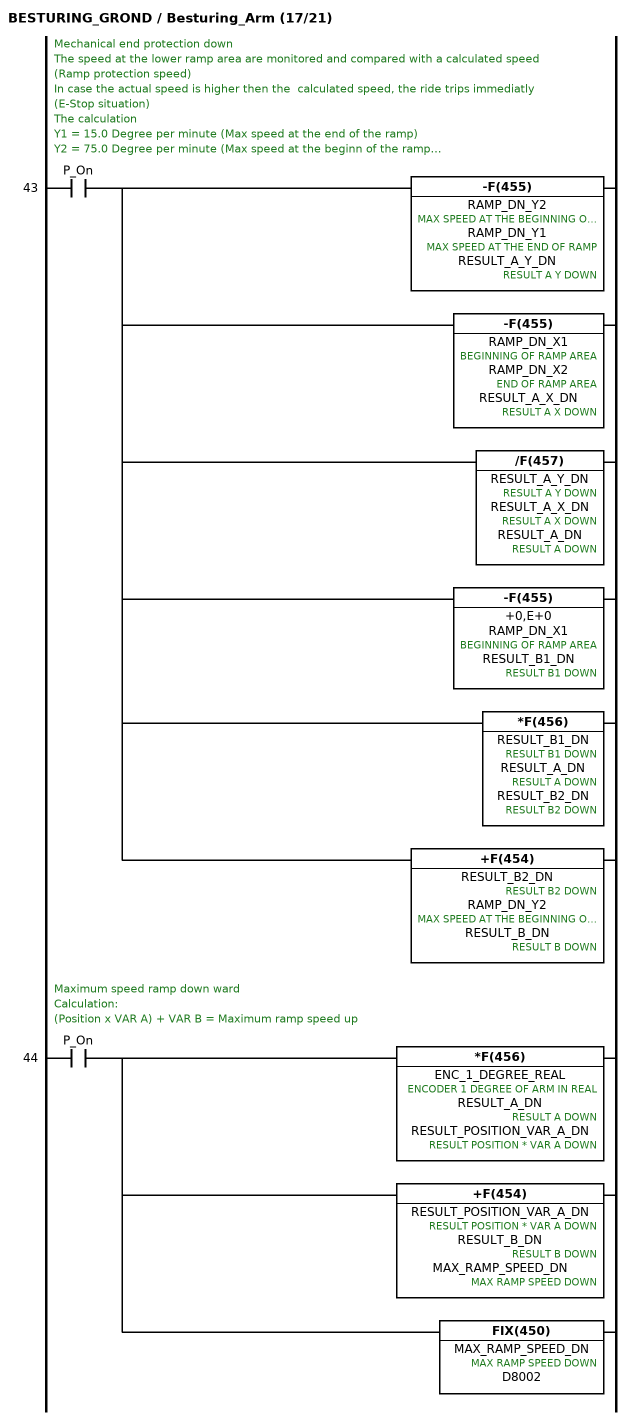
; rung 43: Mechanical end protection down / The speed at the lower ramp area are monitored and compared with a calculated speed (Ramp protection speed) / In case the actual speed is higher then the  calculated speed, the ride trips immediatly (E-Stop situation) / The calculation / Y1 = 15.0 Degree per minute (Max speed at the end of the ramp) / Y2 = 75.0 Degree per minute (Max speed at the beginn of the ramp) / X1 = 8.0 Degree (Begin of ramp area) / X2 = 0.0 Degree (End of ramp area) / The formula for A: / Y2 - Y1 / A =    ------- / X1 - X2 / The formula for B: / B =    (A * (0 - X1) + Y2
LD P_On
-F(455) RAMP_DN_Y2 RAMP_DN_Y1 RESULT_A_Y_DN  ; MAX SPEED AT THE BEGINNING OF RAMP, MAX SPEED AT THE END OF RAMP, RESULT A Y DOWN
-F(455) RAMP_DN_X1 RAMP_DN_X2 RESULT_A_X_DN  ; BEGINNING OF RAMP AREA, END OF RAMP AREA, RESULT A X DOWN
/F(457) RESULT_A_Y_DN RESULT_A_X_DN RESULT_A_DN  ; RESULT A Y DOWN, RESULT A X DOWN, RESULT A DOWN
-F(455) +0,E+0 RAMP_DN_X1 RESULT_B1_DN  ; BEGINNING OF RAMP AREA, RESULT B1 DOWN
*F(456) RESULT_B1_DN RESULT_A_DN RESULT_B2_DN  ; RESULT B1 DOWN, RESULT A DOWN, RESULT B2 DOWN
+F(454) RESULT_B2_DN RAMP_DN_Y2 RESULT_B_DN  ; RESULT B2 DOWN, MAX SPEED AT THE BEGINNING OF RAMP, RESULT B DOWN
; rung 44: Maximum speed ramp down ward / Calculation: / (Position x VAR A) + VAR B = Maximum ramp speed up
LD P_On
*F(456) ENC_1_DEGREE_REAL RESULT_A_DN RESULT_POSITION_VAR_A_DN  ; ENCODER 1 DEGREE OF ARM IN REAL, RESULT A DOWN, RESULT POSITION * VAR A DOWN
+F(454) RESULT_POSITION_VAR_A_DN RESULT_B_DN MAX_RAMP_SPEED_DN  ; RESULT POSITION * VAR A DOWN, RESULT B DOWN, MAX RAMP SPEED DOWN
FIX(450) MAX_RAMP_SPEED_DN D8002  ; MAX RAMP SPEED DOWN

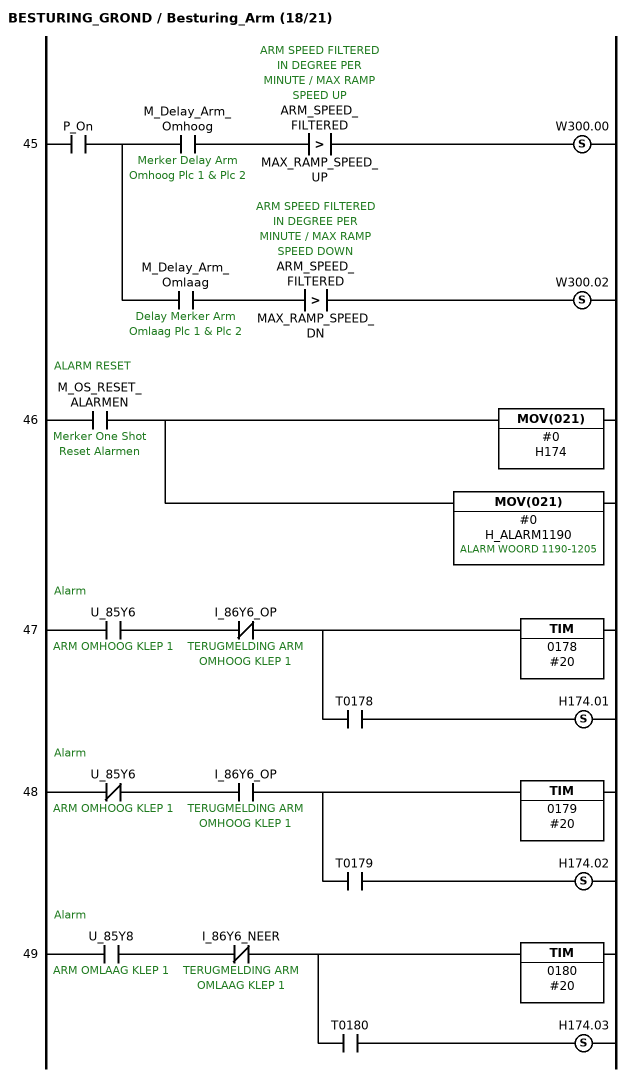
; rung 45
LD P_On
OUT TR0
AND M_Delay_Arm_Omhoog  ; Merker Delay Arm Omhoog Plc 1 & Plc 2
AND>F(333) ARM_SPEED_FILTERED MAX_RAMP_SPEED_UP  ; ARM SPEED FILTERED IN DEGREE PER MINUTE, MAX RAMP SPEED UP
SET W300.00
LD TR0
AND M_Delay_Arm_Omlaag  ; Delay Merker Arm Omlaag Plc 1 & Plc 2
AND>F(333) ARM_SPEED_FILTERED MAX_RAMP_SPEED_DN  ; ARM SPEED FILTERED IN DEGREE PER MINUTE, MAX RAMP SPEED DOWN
SET W300.02
; rung 46: ALARM RESET
LD M_OS_RESET_ALARMEN  ; Merker One Shot Reset Alarmen
MOV(021) #0 H174
MOV(021) #0 H_ALARM1190  ; ALARM WOORD 1190-1205
; rung 47: Alarm
LD U_85Y6  ; ARM OMHOOG KLEP 1
ANDNOT I_86Y6_OP  ; TERUGMELDING ARM OMHOOG KLEP 1
TIM 0178 #20
AND T0178
SET H174.01
; rung 48: Alarm
LDNOT U_85Y6  ; ARM OMHOOG KLEP 1
AND I_86Y6_OP  ; TERUGMELDING ARM OMHOOG KLEP 1
TIM 0179 #20
AND T0179
SET H174.02
; rung 49: Alarm
LD U_85Y8  ; ARM OMLAAG KLEP 1
ANDNOT I_86Y6_NEER  ; TERUGMELDING ARM OMLAAG KLEP 1
TIM 0180 #20
AND T0180
SET H174.03

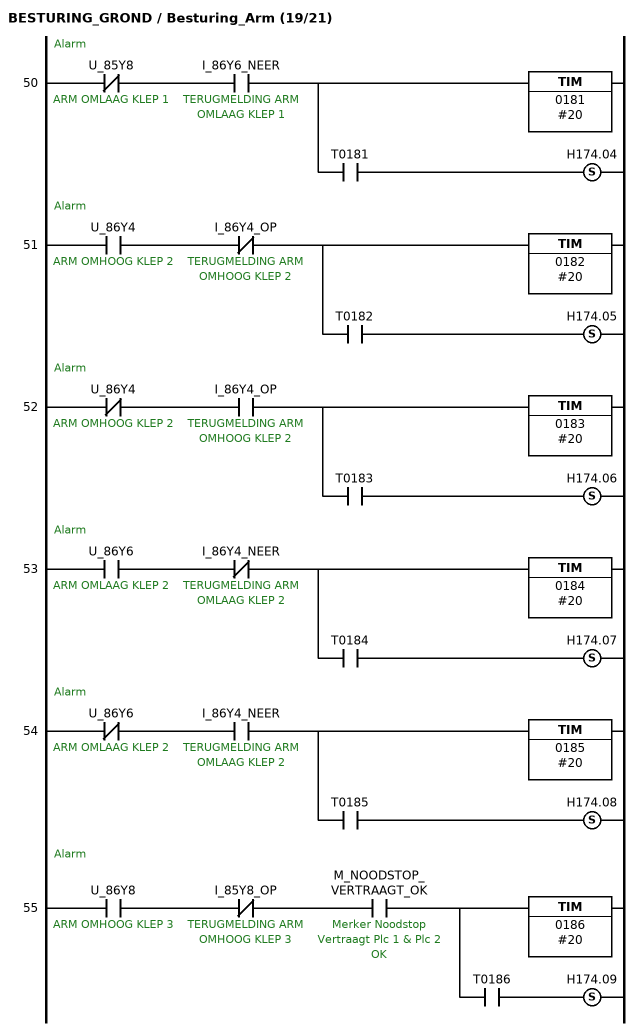
; rung 50: Alarm
LDNOT U_85Y8  ; ARM OMLAAG KLEP 1
AND I_86Y6_NEER  ; TERUGMELDING ARM OMLAAG KLEP 1
TIM 0181 #20
AND T0181
SET H174.04
; rung 51: Alarm
LD U_86Y4  ; ARM OMHOOG KLEP 2
ANDNOT I_86Y4_OP  ; TERUGMELDING ARM OMHOOG KLEP 2
TIM 0182 #20
AND T0182
SET H174.05
; rung 52: Alarm
LDNOT U_86Y4  ; ARM OMHOOG KLEP 2
AND I_86Y4_OP  ; TERUGMELDING ARM OMHOOG KLEP 2
TIM 0183 #20
AND T0183
SET H174.06
; rung 53: Alarm
LD U_86Y6  ; ARM OMLAAG KLEP 2
ANDNOT I_86Y4_NEER  ; TERUGMELDING ARM OMLAAG KLEP 2
TIM 0184 #20
AND T0184
SET H174.07
; rung 54: Alarm
LDNOT U_86Y6  ; ARM OMLAAG KLEP 2
AND I_86Y4_NEER  ; TERUGMELDING ARM OMLAAG KLEP 2
TIM 0185 #20
AND T0185
SET H174.08
; rung 55: Alarm
LD U_86Y8  ; ARM OMHOOG KLEP 3
ANDNOT I_85Y8_OP  ; TERUGMELDING ARM OMHOOG KLEP 3
AND M_NOODSTOP_VERTRAAGT_OK  ; Merker Noodstop Vertraagt Plc 1 & Plc 2 OK
TIM 0186 #20
AND T0186
SET H174.09

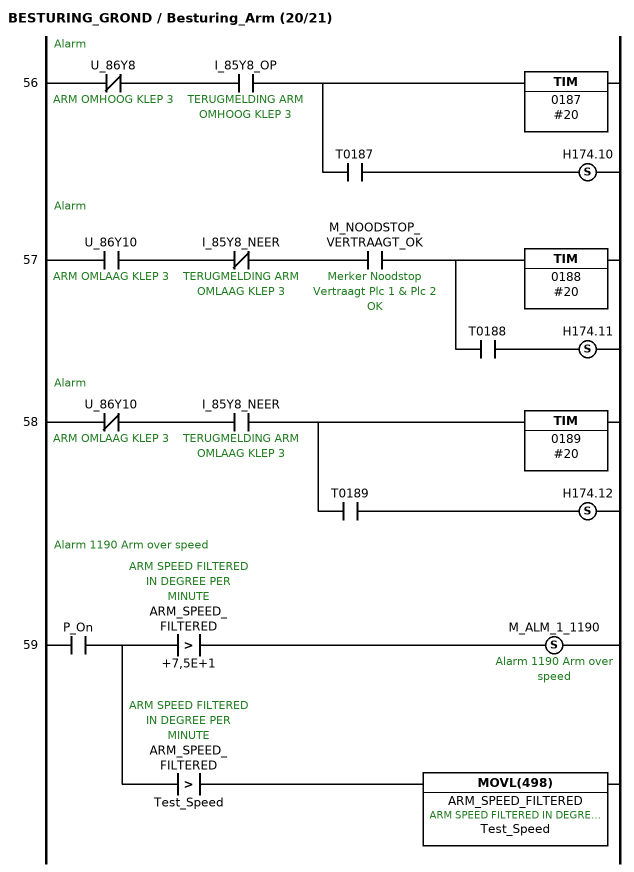
; rung 56: Alarm
LDNOT U_86Y8  ; ARM OMHOOG KLEP 3
AND I_85Y8_OP  ; TERUGMELDING ARM OMHOOG KLEP 3
TIM 0187 #20
AND T0187
SET H174.10
; rung 57: Alarm
LD U_86Y10  ; ARM OMLAAG KLEP 3
ANDNOT I_85Y8_NEER  ; TERUGMELDING ARM OMLAAG KLEP 3
AND M_NOODSTOP_VERTRAAGT_OK  ; Merker Noodstop Vertraagt Plc 1 & Plc 2 OK
TIM 0188 #20
AND T0188
SET H174.11
; rung 58: Alarm
LDNOT U_86Y10  ; ARM OMLAAG KLEP 3
AND I_85Y8_NEER  ; TERUGMELDING ARM OMLAAG KLEP 3
TIM 0189 #20
AND T0189
SET H174.12
; rung 59: Alarm 1190 Arm over speed
LD P_On
OUT TR0
AND>F(333) ARM_SPEED_FILTERED +7,5E+1  ; ARM SPEED FILTERED IN DEGREE PER MINUTE
SET M_ALM_1_1190  ; Alarm 1190 Arm over speed
LD TR0
AND>F(333) ARM_SPEED_FILTERED Test_Speed  ; ARM SPEED FILTERED IN DEGREE PER MINUTE
MOVL(498) ARM_SPEED_FILTERED Test_Speed  ; ARM SPEED FILTERED IN DEGREE PER MINUTE

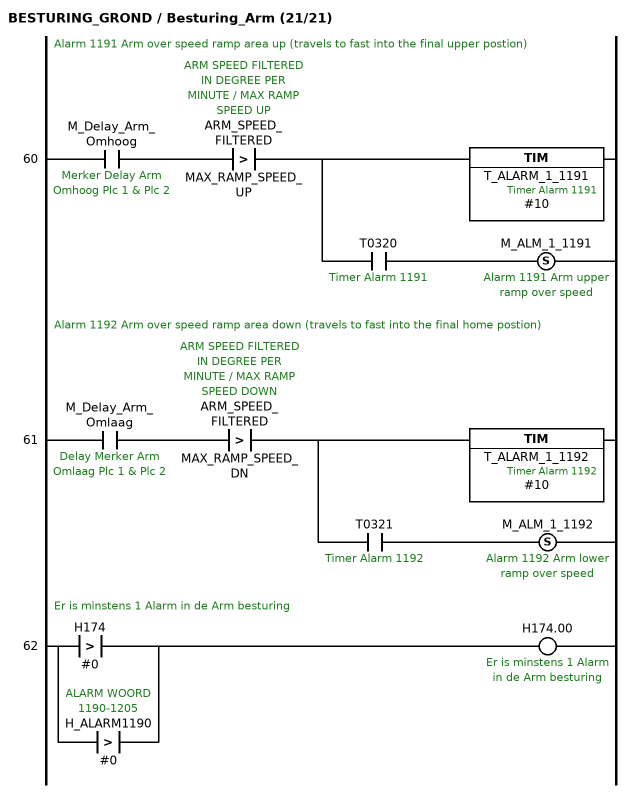
; rung 60: Alarm 1191 Arm over speed ramp area up (travels to fast into the final upper postion)
LD M_Delay_Arm_Omhoog  ; Merker Delay Arm Omhoog Plc 1 & Plc 2
AND>F(333) ARM_SPEED_FILTERED MAX_RAMP_SPEED_UP  ; ARM SPEED FILTERED IN DEGREE PER MINUTE, MAX RAMP SPEED UP
TIM T_ALARM_1_1191 #10  ; Timer Alarm 1191
AND T0320  ; Timer Alarm 1191
SET M_ALM_1_1191  ; Alarm 1191 Arm upper ramp over speed
; rung 61: Alarm 1192 Arm over speed ramp area down (travels to fast into the final home postion)
LD M_Delay_Arm_Omlaag  ; Delay Merker Arm Omlaag Plc 1 & Plc 2
AND>F(333) ARM_SPEED_FILTERED MAX_RAMP_SPEED_DN  ; ARM SPEED FILTERED IN DEGREE PER MINUTE, MAX RAMP SPEED DOWN
TIM T_ALARM_1_1192 #10  ; Timer Alarm 1192
AND T0321  ; Timer Alarm 1192
SET M_ALM_1_1192  ; Alarm 1192 Arm lower ramp over speed
; rung 62: Er is minstens 1 Alarm in de Arm besturing
LD>(320) H174 #0
OR>(320) H_ALARM1190 #0  ; ALARM WOORD 1190-1205
OUT H174.00  ; Er is minstens 1 Alarm in de Arm besturing

### Section Einde_Besturing_Grond
; rung 0
END(001)

## Program SIGNALEN_EILAND (cyclic task 10)

### Section Fast_Counter_Control

### Section Incrementele_Encoder_Decoder_4

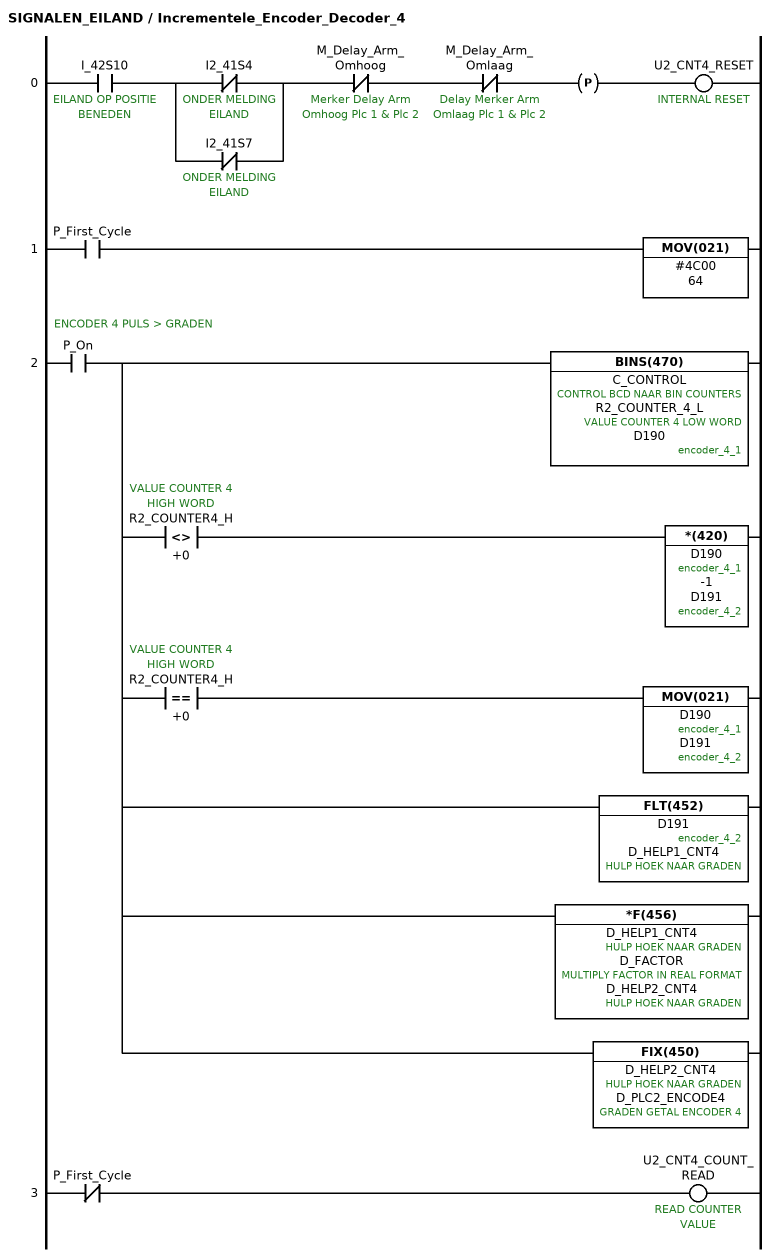
; rung 0
LD I_42S10  ; EILAND OP POSITIE BENEDEN
LDNOT I2_41S4  ; ONDER MELDING EILAND
ORNOT I2_41S7  ; ONDER MELDING EILAND
ANDLD
ANDNOT M_Delay_Arm_Omhoog  ; Merker Delay Arm Omhoog Plc 1 & Plc 2
ANDNOT M_Delay_Arm_Omlaag  ; Delay Merker Arm Omlaag Plc 1 & Plc 2
UP(521)
OUT U2_CNT4_RESET  ; INTERNAL RESET
; rung 1
LD P_First_Cycle
MOV(021) #4C00 64
; rung 2: ENCODER 4 PULS > GRADEN
LD P_On
OUT TR0
BINS(470) C_CONTROL R2_COUNTER_4_L D190  ; CONTROL BCD NAAR BIN COUNTERS, VALUE COUNTER 4 LOW WORD, encoder_4_1
AND<>S(307) R2_COUNTER4_H +0  ; VALUE COUNTER 4 HIGH WORD
*(420) D190 -1 D191  ; encoder_4_1, encoder_4_2
LD TR0
AND=S(302) R2_COUNTER4_H +0  ; VALUE COUNTER 4 HIGH WORD
MOV(021) D190 D191  ; encoder_4_1, encoder_4_2
LD TR0
FLT(452) D191 D_HELP1_CNT4  ; encoder_4_2, HULP HOEK NAAR GRADEN
*F(456) D_HELP1_CNT4 D_FACTOR D_HELP2_CNT4  ; HULP HOEK NAAR GRADEN, MULTIPLY FACTOR IN REAL FORMAT
FIX(450) D_HELP2_CNT4 D_PLC2_ENCODE4  ; HULP HOEK NAAR GRADEN, GRADEN GETAL ENCODER 4
; rung 3
LDNOT P_First_Cycle
OUT U2_CNT4_COUNT_READ  ; READ COUNTER VALUE

### Section Horizon_Decoder_Eiland

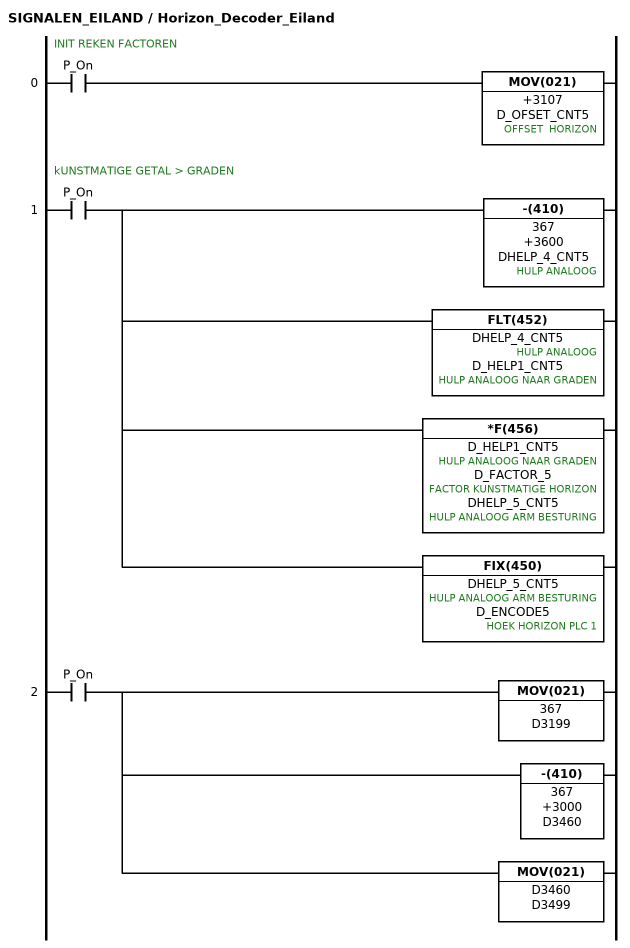
; rung 0: INIT REKEN FACTOREN
LD P_On
MOV(021) +3107 D_OFSET_CNT5  ; OFFSET  HORIZON
; rung 1: kUNSTMATIGE GETAL > GRADEN
LD P_On
-(410) 367 +3600 DHELP_4_CNT5  ; HULP ANALOOG
FLT(452) DHELP_4_CNT5 D_HELP1_CNT5  ; HULP ANALOOG, HULP ANALOOG NAAR GRADEN
*F(456) D_HELP1_CNT5 D_FACTOR_5 DHELP_5_CNT5  ; HULP ANALOOG NAAR GRADEN, FACTOR KUNSTMATIGE HORIZON, HULP ANALOOG ARM BESTURING
FIX(450) DHELP_5_CNT5 D_ENCODE5  ; HULP ANALOOG ARM BESTURING, HOEK HORIZON PLC 1
; rung 2
LD P_On
MOV(021) 367 D3199
-(410) 367 +3000 D3460
MOV(021) D3460 D3499

### Section Controle_Positie_Eiland

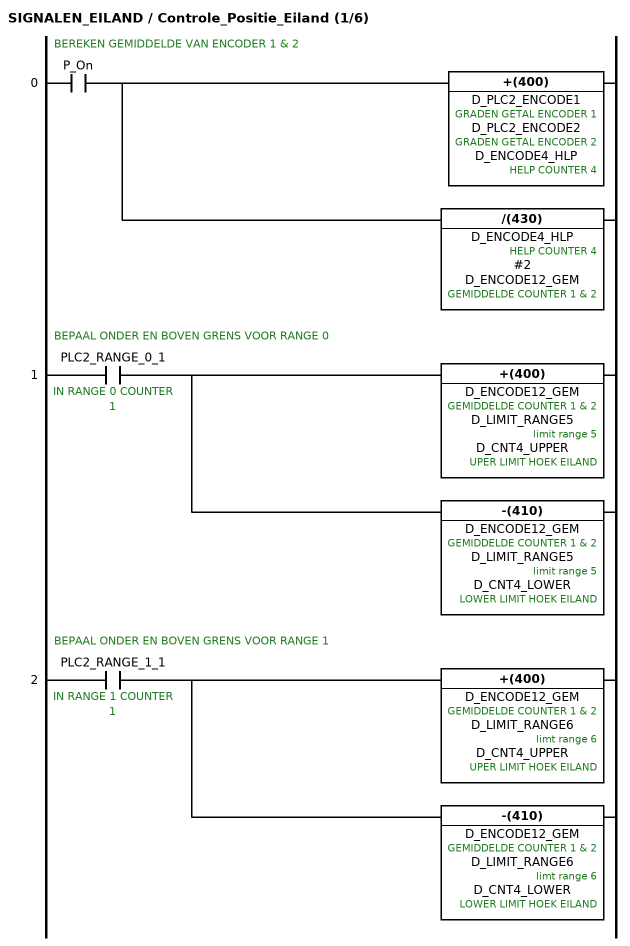
; rung 0: BEREKEN GEMIDDELDE VAN ENCODER 1 & 2
LD P_On
+(400) D_PLC2_ENCODE1 D_PLC2_ENCODE2 D_ENCODE4_HLP  ; GRADEN GETAL ENCODER 1, GRADEN GETAL ENCODER 2, HELP COUNTER 4
/(430) D_ENCODE4_HLP #2 D_ENCODE12_GEM  ; HELP COUNTER 4, GEMIDDELDE COUNTER 1 & 2
; rung 1: BEPAAL ONDER EN BOVEN GRENS VOOR RANGE 0
LD PLC2_RANGE_0_1  ; IN RANGE 0 COUNTER 1
+(400) D_ENCODE12_GEM D_LIMIT_RANGE5 D_CNT4_UPPER  ; GEMIDDELDE COUNTER 1 & 2, limit range 5, UPER LIMIT HOEK EILAND
-(410) D_ENCODE12_GEM D_LIMIT_RANGE5 D_CNT4_LOWER  ; GEMIDDELDE COUNTER 1 & 2, limit range 5, LOWER LIMIT HOEK EILAND
; rung 2: BEPAAL ONDER EN BOVEN GRENS VOOR RANGE 1
LD PLC2_RANGE_1_1  ; IN RANGE 1 COUNTER 1
+(400) D_ENCODE12_GEM D_LIMIT_RANGE6 D_CNT4_UPPER  ; GEMIDDELDE COUNTER 1 & 2, limt range 6, UPER LIMIT HOEK EILAND
-(410) D_ENCODE12_GEM D_LIMIT_RANGE6 D_CNT4_LOWER  ; GEMIDDELDE COUNTER 1 & 2, limt range 6, LOWER LIMIT HOEK EILAND

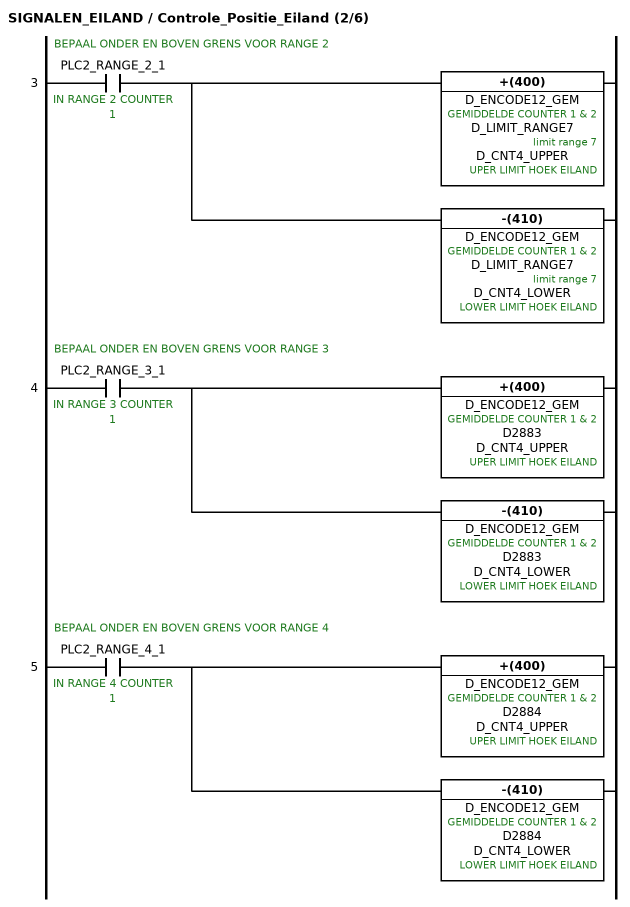
; rung 3: BEPAAL ONDER EN BOVEN GRENS VOOR RANGE 2
LD PLC2_RANGE_2_1  ; IN RANGE 2 COUNTER 1
+(400) D_ENCODE12_GEM D_LIMIT_RANGE7 D_CNT4_UPPER  ; GEMIDDELDE COUNTER 1 & 2, limit range 7, UPER LIMIT HOEK EILAND
-(410) D_ENCODE12_GEM D_LIMIT_RANGE7 D_CNT4_LOWER  ; GEMIDDELDE COUNTER 1 & 2, limit range 7, LOWER LIMIT HOEK EILAND
; rung 4: BEPAAL ONDER EN BOVEN GRENS VOOR RANGE 3
LD PLC2_RANGE_3_1  ; IN RANGE 3 COUNTER 1
+(400) D_ENCODE12_GEM D2883 D_CNT4_UPPER  ; GEMIDDELDE COUNTER 1 & 2, UPER LIMIT HOEK EILAND
-(410) D_ENCODE12_GEM D2883 D_CNT4_LOWER  ; GEMIDDELDE COUNTER 1 & 2, LOWER LIMIT HOEK EILAND
; rung 5: BEPAAL ONDER EN BOVEN GRENS VOOR RANGE 4
LD PLC2_RANGE_4_1  ; IN RANGE 4 COUNTER 1
+(400) D_ENCODE12_GEM D2884 D_CNT4_UPPER  ; GEMIDDELDE COUNTER 1 & 2, UPER LIMIT HOEK EILAND
-(410) D_ENCODE12_GEM D2884 D_CNT4_LOWER  ; GEMIDDELDE COUNTER 1 & 2, LOWER LIMIT HOEK EILAND

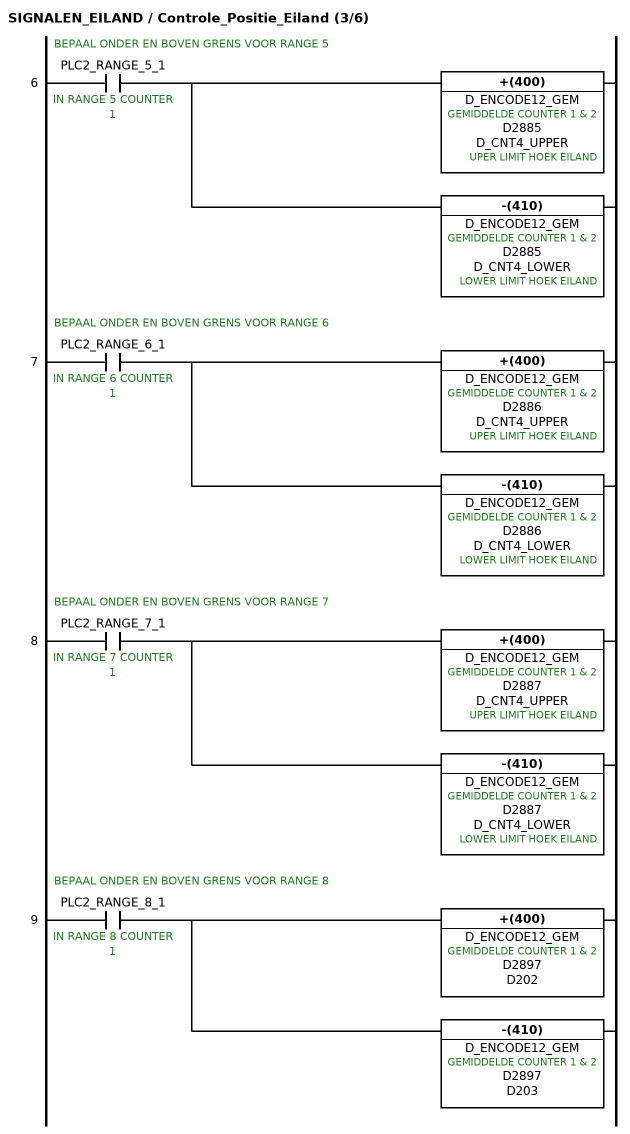
; rung 6: BEPAAL ONDER EN BOVEN GRENS VOOR RANGE 5
LD PLC2_RANGE_5_1  ; IN RANGE 5 COUNTER 1
+(400) D_ENCODE12_GEM D2885 D_CNT4_UPPER  ; GEMIDDELDE COUNTER 1 & 2, UPER LIMIT HOEK EILAND
-(410) D_ENCODE12_GEM D2885 D_CNT4_LOWER  ; GEMIDDELDE COUNTER 1 & 2, LOWER LIMIT HOEK EILAND
; rung 7: BEPAAL ONDER EN BOVEN GRENS VOOR RANGE 6
LD PLC2_RANGE_6_1  ; IN RANGE 6 COUNTER 1
+(400) D_ENCODE12_GEM D2886 D_CNT4_UPPER  ; GEMIDDELDE COUNTER 1 & 2, UPER LIMIT HOEK EILAND
-(410) D_ENCODE12_GEM D2886 D_CNT4_LOWER  ; GEMIDDELDE COUNTER 1 & 2, LOWER LIMIT HOEK EILAND
; rung 8: BEPAAL ONDER EN BOVEN GRENS VOOR RANGE 7
LD PLC2_RANGE_7_1  ; IN RANGE 7 COUNTER 1
+(400) D_ENCODE12_GEM D2887 D_CNT4_UPPER  ; GEMIDDELDE COUNTER 1 & 2, UPER LIMIT HOEK EILAND
-(410) D_ENCODE12_GEM D2887 D_CNT4_LOWER  ; GEMIDDELDE COUNTER 1 & 2, LOWER LIMIT HOEK EILAND
; rung 9: BEPAAL ONDER EN BOVEN GRENS VOOR RANGE 8
LD PLC2_RANGE_8_1  ; IN RANGE 8 COUNTER 1
+(400) D_ENCODE12_GEM D2897 D202  ; GEMIDDELDE COUNTER 1 & 2
-(410) D_ENCODE12_GEM D2897 D203  ; GEMIDDELDE COUNTER 1 & 2

